// TIA Portal V17 export
// export: Created 2025-04-14T02:57:49.6902686Z, ExportSetting WithDefaults, DisplayName Totally Integrated Automation Portal, DisplayVersion V17, DisplayName TIA Portal Openness, DisplayVersion V17, DisplayName TIA Portal Version Control Interface, DisplayVersion V17, DisplayName SINAMICS Startdrive Advanced, DisplayVersion V17, DisplayName SINAMICS Startdrive G130, G150, S120, S150, SINAMICS MV, S210, DisplayVersion V17, DisplayName SINAMICS Startdrive G110M, G120, G120C, G120D, G120P, G115D, DisplayVersion V17, DisplayName STEP 7 Professional, DisplayVersion V17, DisplayName STEP 7 Safety, DisplayVersion V17, DisplayName WinCC Advanced, DisplayVersion V17
TYPE "UDT_Modbus_ALM"
// stored: IsFailsafeCompliant false
   STRUCT
      ModbusStatus : Word;   // Modbus通信状态/错误码
      ConversionError : Word;   // 数据转换错误码
      DeserializeStatus : Word;   // 反序列化状态/错误码
   END_STRUCT;
END_TYPE
